// TIA Portal V18 export
DATA_BLOCK "Function recirculation"   // DB76
{ S7_Optimized_Access := 'TRUE' }
VERSION : 0.1
// stored: AutoNumber true, DBAccessibleFromOPCUA true, IsOnlyStoredInLoadMemory false, IsRetainMemResEnabled false, IsWriteProtectedInAS false, MemoryReserve 100
   VAR RETAIN
      Selection : Struct
         "A" : Int;
         "B" : Int;
         "A A AB" : Int;
         "A selected" : Bool;
         "B selected" : Bool;
         "A or B selected" : Bool;
      END_STRUCT;
      "recirculation method" : Struct
         "A" : Int;
         "B" : Int;
         "A with Pump" : Bool;
         "B with Pump" : Bool;
         "A or B with Pump" : Bool;
         "A without Pump selected" : Bool;
         "B without Pump selected" : Bool;
      END_STRUCT;
      "time" : Struct
         "active time" : Int;
         "idle time" : Int;
      END_STRUCT;
      Flowrate : Struct
         "A" : Real;
         "B" : Real;
      END_STRUCT;
   END_VAR
   VAR
      "Control A" : Struct
         "start A1" : Bool;
         "start A2" : Bool;
      END_STRUCT;
      "Control B" : Struct
         "start B" : Bool;
      END_STRUCT;
      "Output A1" : Struct
         "ON recirculation valve" : Bool;
         "ON pump" : Bool;
         "On time Done" : Bool;
         Running : Bool;
         Blink : Bool;
      END_STRUCT;
      "Output A2" : Struct
         "ON recirculation valve" : Bool;
         "ON pump" : Bool;
         "On time Done" : Bool;
         Running : Bool;
         Blink : Bool;
      END_STRUCT;
      "Output B1" : Struct
         "ON recirculation valve" : Bool;
         "On time Done" : Bool;
         "ON pump" : Bool;
         Running : Bool;
         Blink : Bool;
      END_STRUCT;
      "time in sec" : Struct
         "active time" : DInt;
         "idle time" : DInt;
      END_STRUCT;
      "A1 time PV" : Struct
         "Active time PV" : Int;
         "Active time PV_ms" : DInt;
         "IDLE time PV_ms" : DInt;
         "IDLE time PV" : Int;
      END_STRUCT;
      "A2 time PV" : Struct
         "Active time PV" : Int;
         "Active time PV_ms" : DInt;
         "IDLE time PV_ms" : DInt;
         "IDLE time PV" : Int;
      END_STRUCT;
      "B1 time PV" : Struct
         "Active time PV" : Int;
         "Active time PV_ms" : DInt;
         "IDLE time PV_ms" : DInt;
         "IDLE time PV" : Int;
      END_STRUCT;
      "AD-HMI A" : Struct
         "set time" : Int;
         "Time PV" : Int;
         "Blink timer" : Bool;
      END_STRUCT;
      "AD-HMI B" : Struct
         "set time" : Int;
         "Time PV" : Int;
         "Blink timer" : Bool;
      END_STRUCT;
   END_VAR
BEGIN
END_DATA_BLOCK
